// TIA Portal V17 export
// export: Created 2026-04-13T11:12:42.5952848Z, ExportSetting WithDefaults, DisplayName Totally Integrated Automation Portal, DisplayVersion V17 Update 4, DisplayName TIA Portal Openness, DisplayVersion V17 Update 4, DisplayName TIA Portal Version Control Interface, DisplayVersion V17, DisplayName SINAMICS Startdrive Advanced, DisplayVersion V17, DisplayName SINAMICS Startdrive G130, G150, S120, S150, SINAMICS MV, S210, DisplayVersion V17, DisplayName SINAMICS Startdrive G110M, G120, G120C, G120D, G120P, G115D, DisplayVersion V17, DisplayName STEP 7 Professional, DisplayVersion V17 Update 4, DisplayName STEP 7 Safety, DisplayVersion V17, DisplayName WinCC Professional, DisplayVersion V17 Update 4
FUNCTION_BLOCK "6-系统时间读取与设置"   // FB3009, LAD
{ S7_Optimized_Access := 'FALSE' }
VERSION : 0.1
// stored: AutoNumber true, IsIECCheckEnabled false, SetENOAutomatically false, UDAEnableTagReadback false
   VAR_INPUT
      系统时间设置 : Bool;   // 时间设置按钮
      要写入的系统时间 : Date_And_Time := DT#2022-07-27-00:00:00;   // 设定时间
   END_VAR
   VAR_OUTPUT
      系统时间 : Date_And_Time;   // 系统时间
      Year : Byte;   // 年
      Month : Byte;   // 月
      Day : Byte;   // 日
      Hour : Byte;   // 时
      Minute : Byte;   // 分
      Second : Byte;   // 秒
   END_VAR
   VAR DB_SPECIFIC
      SetTimeTP1 : Byte;
      SetTimeTP2 : Byte;
      SetTimeTP3 : Byte;
      SetTimeTP4 : Byte;
      SetTimeTP5 : Byte;
      SetTimeTP6 : Byte;
      SetTimeTP7 : Byte;
      SetTimeTP8 : Byte;
      SetTimeTP9 : Date;
      SetTimeTP10 : Time_Of_Day;
   END_VAR
   VAR_TEMP
      Ret : Int;
   END_VAR
BEGIN

REGION Network 1: 读出系统时间
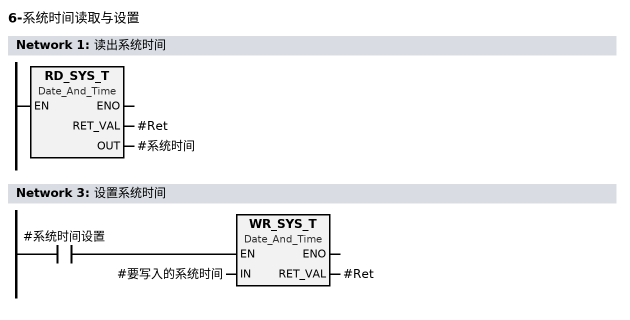
   RUNG wire#powerrail
      { S7_Templates := "date_type := Date_And_Time" } RD_SYS_T(RET_VAL => #Ret, OUT => #系统时间)
   END_RUNG
   // the same network as SCL:
   #Ret := RD_SYS_T(OUT => #系统时间);
END_REGION

NETWORK
TITLE = 读取时间

      L     %DIB10;
      T     #Year;
      L     %DIB11;
      T     #Month;
      L     %DIB12;
      T     #Day;
      L     %DIB13;
      T     #Hour;
      L     %DIB14;
      T     #Minute;
      L     %DIB15;
      T     #Second;


REGION Network 3: 设置系统时间
   RUNG wire#powerrail
      Contact( #系统时间设置 )
      { S7_Templates := "date_type := Date_And_Time" } WR_SYS_T(IN := #要写入的系统时间, RET_VAL => #Ret)
   END_RUNG
   // the same network as SCL:
   IF #系统时间设置 THEN #Ret := WR_SYS_T(IN := #要写入的系统时间); END_IF;
END_REGION
END_FUNCTION_BLOCK
